{attribute 'qualified_only'}
VAR_GLOBAL
    // One PLC-wide clock-quality authority. Hidden here; each root republishes
    // the validated value beside its system-health surface.
    {attribute 'OPC.UA.DA' := '0'}
    Current : ST_TimeQuality;
END_VAR

(* stored: Version 1.1.0.1, ProductVersion 3.1.4024.12
   GVL GVL_FraktalTime: Id {aa7cfe4d-f1fc-4fe8-b319-f1eabed60747} *)
